Universal Robots PolyScope program: OnRobot_Box_Insertion_Example.urp

Program OnRobot_Box_Insertion_Example (createdIn=3.3.4.310 lastSavedIn=3.7.0.40195 robotSerialNumber=2014359999 directory=/home/ur/ursim-current/programs/TransferVM/Examples/Pendrive installation=default)
Calibrated DH parameters: a=[0.000125, -0.611383, -0.570393, -0.000092, 0.000088, 0]; d=[0.127903, 2.433032, -6.959421, 4.690192, 0.11563, 0.092223]; alpha=[1.570378, -0.01465, -0.007405, 1.570477, -1.570381, 0]; deltaTheta=[-0.000064, -0.058226, 0.116976, -0.058728, 0.000029, -0.000013]
BeforeStart
  URCap F/T Zero (FT-OnRobot, OnRobot A/S)
Robot Program (runOnlyOnce=true)
  URCap F/T Guard (FT-OnRobot, OnRobot A/S) dataModel(OF_PID=0, FX=0.0, FY=0.0, FZ=0.0, TX=0.0, TY=0.0, TZ=0.0, F3D=75.0, T3D=2.0, ABS=true, COORD=0, INDEX=0, STATE=true, ADVANCED=false, NEEDDIGI=false, NAME=75N & 2Nm, absolute=true)
    MoveJ speed 60 deg/s, acceleration 80 deg/s^2 (useActiveTCP=false)
      Waypoint StartWP: TCP in base x=-120.113 y=-431.763 z=146.073 mm, rx=-0.0012 ry=3.1163 rz=0.0389 rad; joints [-91.713, -98.956, -126.223, -46.295, 91.393, -1.776] deg
    URCap F/T Insert Box (FT-OnRobot, OnRobot A/S) dataModel(X=0.0, Y=0.0, Z=-0.025, X2=0.0, Y2=0.0, Z2=0.0, RX=-0.2617993877991494, RY=0.0, Rz=0.0, COORD=0, LEN=2, LEN2=0, LEN3=2, DEG=0, SPEED=0.01, ACC=1.2, BREAK=2.0, SILENT=false, DEPTH=0.03, FLIMIT=6.0, TLIMIT=1.0, FMULTI=2.0, x=0.01, y=0.0, z=0.0, x2=0.0, y2=0.0, z2=0.0, rx=0.2617995, ry=0.0, rz=0.0)
    URCap F/T Move (FT-OnRobot, OnRobot A/S) dataModel(coordsys=1, absolute=false, speed=0.03, acceleration=0.5, rpy=[0.0, 0.0, 0.0], popupLimit=false, ftarray=[0.0, 0.0, 0.0, 0.0, 0.0, 0.0, 30.0, 0.0], ftabsarray=[false, false, false, false, false, false])
      URCap F/T Waypoint (FT-OnRobot, OnRobot A/S) dataModel(relativeCoords=[0.0, 0.0, 0.05, 0.0, 0.0, 0.0], type=2, z=-0.02)
